Yaskawa INFORM job: FTP_TEST.JBI

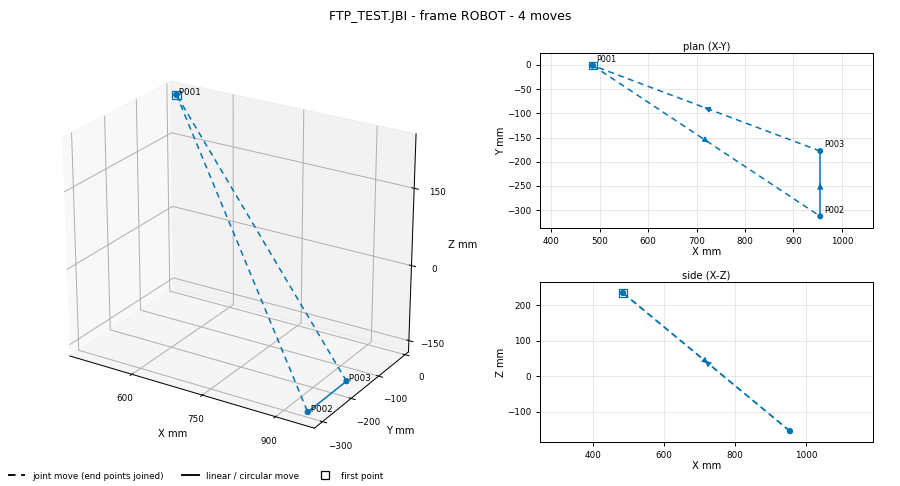
[picture p0: tool path of FTP_TEST.JBI in frame ROBOT, 4 of 5 moves have a stored position in this frame; points joined in program order, loops and branches not executed]
/JOB
//NAME FTP_TEST
//POS
///NPOS 0,0,0,4,0,0
///TOOL 0
///POSTYPE PULSE
///PULSE
P00000=0,0,0,0,0,0
///TOOL 5
///POSTYPE ROBOT
///RECTAN
///RCONF 0,0,0,0,0,0,0,0,0,0,0,0,0,0,0,0,0,0,0,0,0,0,0,0
P00001=485.364,-1.213,234.338,179.9840,20.2111,1.6879
P00002=955.326,-312.783,-154.686,-168.3765,-2.9339,7.0523
P00003=955.326,-178.005,-154.700,-168.3718,-2.9293,7.0363
//INST
///DATE 2024/03/06 12:07
///ATTR SC,RW
///GROUP1 RB1
NOP
MOVJ P001 VJ=5.00
MOVJ P002 VJ=5.00
MOVL P003 V=1.7
MOVJ P001 VJ=4.00
MOVJ P000 VJ=5.00
END
